{attribute 'qualified_only'}
VAR_GLOBAL
	EM: ARRAY[1..5] OF RTU_EM;
END_VAR

(* stored: Version 1.1.0.1, ProductVersion 3.1.4024.12
   GVL GVL_EM: Id {d3796aaf-5534-4af0-88c9-047c2569b44a} *)
